// TIA Portal V21 export
VAR_GLOBAL   // PLC tag table "K_Sequenze_SterilizzatoreTubo"
END_VAR
